// TIA Portal V18 export
TYPE "UDT_PLCtoMES_ext"
// stored: IsFailsafeCompliant false
   STRUCT
      Cmd : Struct
         "PLC.Load_ChickIn" : Bool;   // 查询事件触发位/Loading part process - Components barcodes are ready and request to read
         "PLC.Load_1" : Bool;   // Loading part process - Spare
         "PLC.Load_2" : Bool;   // Loading part process - Spare
         "PLC.Load_3" : Bool;   // Loading part process - Spare
         "PLC.Unload_DataSave" : Bool;   // 结果准备好并要求存储/Unloading part process - Results are ready and request to store
         "PLC.Unload_1" : Bool;   // Unloading part process - Spare
         "PLC.Unload_2" : Bool;   // Unloading part process - Spare
         "PLC.Unload_3" : Bool;   // Unloading part process - Spare
         "PLC.Spare8" : Bool;   // Spare - Future applications
         "PLC.Spare9" : Bool;   // Spare - Future applications
         "PLC.Spare10" : Bool;   // Spare - Future applications
         "PLC.Spare11" : Bool;   // Spare - Future applications
         "PLC.Spare12" : Bool;   // Spare - Future applications
         "PLC.Spare13" : Bool;   // Spare - Future applications
         "PLC.Spare14" : Bool;   // Spare - Future applications
         "PLC.Spare15" : Bool;   // PLC心跳PLC TO MES Heartbeat signal
      END_STRUCT;
   END_STRUCT;
END_TYPE
